TYPE DS_WeberMulFreqSwitching :
STRUCT
	bFreqSwitchingPB_TS : BOOL;
	bFreqRange4080120En : BOOL;
	bFreqRange2550En : BOOL;
	bDisableMultiFreq80kHz : BOOL;
	bDisableMultiFreq40kHz : BOOL;
	iFreqOutput_TS : INT;
END_STRUCT
END_TYPE

(* stored: Version 1.1.0.1, ProductVersion 3.1.4024.12
   DUT DS_WeberMulFreqSwitching: Id {e459ba85-fa07-428f-a1d6-5a0f0f0eb70d} *)
